TYPE DEBUG_STATE :
STRUCT
	bActivate, bCleanup, bConfigure, bDeactivate, bDestroy, bShutdown, bReset : BOOL;
END_STRUCT
END_TYPE

(* stored: Version 1.1.0.1, ProductVersion 3.1.4026.18
   DUT DEBUG_STATE: Id {1cbb488f-2f81-462f-93ff-8ac56b0207f6} *)
